SUBAPPLICATION AX_SUBSCRIBE_BG3_WEB_OPC (* OPC-UA Remote-Subscribe + VT-Hintergrundfarbe auf SoftKey UND AuxFunction2 + lokaler Web-Republish (generisch, ein Kanal) *)
  (* Standard: 61499-2; Description: Copyright (c) 2026 Meisterschulen am Ostbahnhof This program and the accompanying materials are made available under the terms of the Eclipse Public License 2.0 which is available at https://www.eclipse.org/legal/epl-2.0/ SPDX-License-Identifier: EPL-2.0 *)
  (* Version 1.0, 2026-09-07, Franz Höpfinger, Meisterschulen am Ostbahnhof, Aus Softkey_Aux_IXA_TO_Remote_WRITE_BG_OPC herausgeloest: nur die Status-Seite (Remote-Subscribe + Hintergrundfarbe SoftKey+Aux + lokaler Web-Republish) *)
  PACKAGE MyLib::sys;
  IMPORT isobus::UT::Q::const::IDs::ID_NULL;
  (* Documentation:
  Remote-Subscribe → Hintergrundfarbe (SoftKey+Aux) + lokaler Web-Republish
   Status-Haelfte von Softkey_Aux_IXA_TO_Remote_WRITE_BG_OPC, herausgeloest als eigener Baustein - Erweiterung von AX_SUBSCRIBE_BG_OPC (Subscribe + einfache Hintergrundfarbe) um zwei Dinge:
    - GreenWhiteBackground3_AX statt GreenWhiteBackground1_AX - faerbt sowohl einen SoftKey (u16ObjId) als auch eine AuxFunction2 (u16ObjIdA) synchron.
   - AX_SPLIT_2 spiegelt den empfangenen Zustand zusaetzlich ueber STATUS_WEB_PUBLISH (ID_STATUS_WEB) auf den lokalen OPC-UA-Server DIESES Moduls - ein Web-Client (z.B. vt-ui-mirror), der nur mit diesem Modul verbunden ist, kann so denselben Status lesen, den das echte VT als Hintergrundfarbe zeigt, ohne selbst eine Verbindung zum Zielmodul aufzubauen.
    Fuer nur einen SoftKey ohne Aux AX_SUBSCRIBE_BG_OPC verwenden (kein Web-Republish). Fuer die komplette, vorverdrahtete Kombination mit der Kommando-Seite weiterhin Softkey_Aux_IXA_TO_Remote_WRITE_BG_OPC verwenden.
  *)
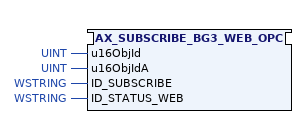
  VAR_INPUT
    u16ObjId : UINT := ID_NULL; (* Object ID SoftKey/Hintergrund (VT) *)
    u16ObjIdA : UINT := ID_NULL; (* Object ID AuxFunction2/Hintergrund (VT) *)
    ID_SUBSCRIBE : WSTRING; (* Remote-Subscribe-Adresse (Status/Farbe, ACTION=SUBSCRIBE) *)
    ID_STATUS_WEB : WSTRING; (* Lokale Publish-Adresse (auf diesem Modul) fuer den vom Zielmodul zurueckgemeldeten Zustand - damit ein Web-Client (z.B. vt-ui-mirror) dieselbe Hintergrundfarbe wie das echte VT zeigen kann *)
  END_VAR
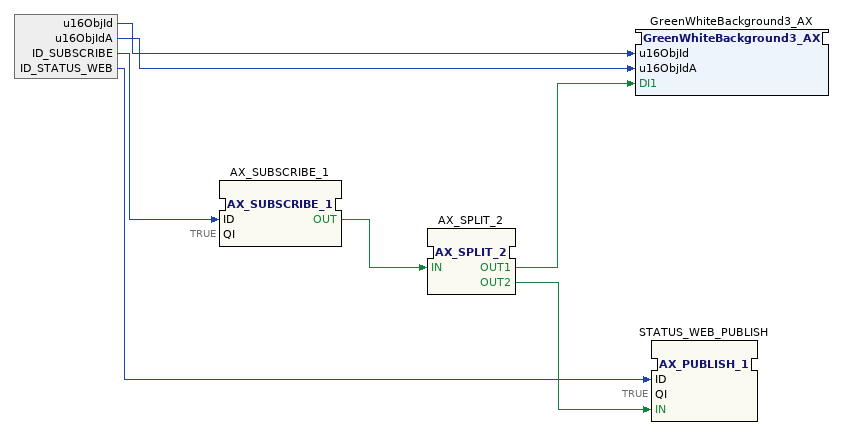
  FBS
    AX_SUBSCRIBE_1 : adapter::net::AX_SUBSCRIBE_1(QI := TRUE);
    AX_SPLIT_2 : adapter::events::unidirectional::AX_SPLIT_2;
    STATUS_WEB_PUBLISH : adapter::net::AX_PUBLISH_1(QI := TRUE);
  END_FBS
  SUBAPPS
    GreenWhiteBackground3_AX : MyLib::sys::GreenWhiteBackground3_AX;
  END_SUBAPPS
  DATA_CONNECTIONS
    u16ObjId TO GreenWhiteBackground3_AX.u16ObjId;
    u16ObjIdA TO GreenWhiteBackground3_AX.u16ObjIdA;
    ID_SUBSCRIBE TO AX_SUBSCRIBE_1.ID;
    ID_STATUS_WEB TO STATUS_WEB_PUBLISH.ID;
  END_CONNECTIONS
  ADAPTER_CONNECTIONS
    AX_SUBSCRIBE_1.OUT TO AX_SPLIT_2.IN;
    AX_SPLIT_2.OUT1 TO GreenWhiteBackground3_AX.DI1;
    AX_SPLIT_2.OUT2 TO STATUS_WEB_PUBLISH.IN;
  END_CONNECTIONS
END_SUBAPPLICATION
